// TIA Portal project "Training" (V13)

(* hardware
DEVICE "S71500/ET200MP station_1"  S7-1500 station
   slot 0: "Rail_0"  6ES7 590-1***0-0AA0
   slot 1: "PLC_1"  CPU 1516F-3 PN/DP  6ES7 516-3FN00-0AB0  V1.7
   slot 2: "DI 16x24VDC HF_1"  DI 16x24VDC HF  6ES7 521-1BH00-0AB0  V2.0
   slot 3: "AI 8xU/I/RTD/TC ST_1"  AI 8xU/I/RTD/TC ST  6ES7 531-7KF00-0AB0  V2.0
   slot 4: "CP 1543-1_1"  CP 1543-1  6GK7 543-1AX00-0XE0  V1.1
DEVICE "ET 200SP station_1"  ET 200SP-Station
   slot 0: "Rack_0"  6ES5 710-8MAx1
   slot 0: "IO device_1"  IM155-6 PN ST  6ES7 155-6AU00-0BN0  V3.1
   slot 1: "AQ 4xU/I ST_1"  AQ 4xU/I ST  6ES7 135-6HD00-0BA1  V1.0
      slot 1: "AQ 4xU/I ST_1"  AQ 4xU/I ST  6ES7 135-6HD00-0BA1
   slot 2: "DQ 16x24VDC/0.5A ST_1"  DQ 16x24VDC/0.5A ST  6ES7 132-6BH00-0BA0  V1.0
      slot 1: "DQ 16x24VDC/0.5A ST_1"  DQ 16x24VDC/0.5A ST  6ES7 132-6BH00-0BA0
   slot 3: "RQ 4x120VDC/230VAC/5A NO ST_1"  DQ 4x24VDC/2A ST  6ES7 132-6HD00-0BB0  V1.1
      slot 1: "RQ 4x120VDC/230VAC/5A NO ST_1"  RQ 4x120VDC/230VAC/5A NO ST  6ES7 132-6HD00-0BB0
   slot 4: "Server module_1"  Server module  6ES7 193-6PA00-0AA0  V1.0
      slot 1: "Server module_1"  Server module  6ES7 193-6PA00-0AA0
   slot 127: "PROFINET BusAdapter CU"  PROFINET Interface  6ES7 193-6AR00-0AA0  V0.0
      slot 1: "Port_1"  6ES7 193-6AR00-0AA0  V0.0
      slot 2: "Port_2"  6ES7 193-6AR00-0AA0  V0.0
DEVICE "KP8_1"  SIMATIC Key Panel
   slot 0: "Rack"  Rail  V1.0
   slot 0: "KP8_1"  KP8  6AV3 688-3AY36-0AX0  R01.00.00
DEVICE "S7-1200 station_1"  S7-1200 Station
   slot 0: "Rack_0"  Rack  V1.0
   slot 1: "PLC_2"  CPU 1215C AC/DC/Rly  6ES7 215-1BG40-0XB0  V4.1
*)

// ===== PLC "PLC_1"  CPU 1516F-3 PN/DP =====

VAR_GLOBAL   // PLC tag table "Default tag table"
   "System_Byte" AT %MB1 : Byte;
   "FirstScan" AT %M1.0 : Bool;
   "DiagStatusUpdate" AT %M1.1 : Bool;
   "AlwaysTRUE" AT %M1.2 : Bool;
   "AlwaysFALSE" AT %M1.3 : Bool;
   "Clock_Byte" AT %MB0 : Byte;
   "Clock_10Hz" AT %M0.0 : Bool;
   "Clock_5Hz" AT %M0.1 : Bool;
   "Clock_2.5Hz" AT %M0.2 : Bool;
   "Clock_2Hz" AT %M0.3 : Bool;
   "Clock_1.25Hz" AT %M0.4 : Bool;
   "Clock_1Hz" AT %M0.5 : Bool;
   "Clock_0.625Hz" AT %M0.6 : Bool;
   "Clock_0.5Hz" AT %M0.7 : Bool;
   "Latch Output" AT %Q50.0 : Bool;
   "Indicated Deg C_1" AT %MW2 : Int;
   "Indicated Deg c_2" AT %MW4 : Int;
   "Run Status" AT %M6.0 : Bool;
   "Counter Reset Bit" AT %M6.1 : Bool;
   "Motor 1 Running" AT %M6.2 : Bool;
   "Motor 2 Running" AT %M6.3 : Bool;
   "Outputs to Transfer Area" AT %QB100 : Byte;
   "Inputs from Transfer Area" AT %IB100 : Byte;
   "Clock Byte Data from 1200" AT %MB100 : Byte;
END_VAR

VAR_GLOBAL   // PLC tag table "Local IO Tags"
   "S71500 Green PB" AT %I0.0 : Bool;
   "S71500 Blue PB" AT %I0.1 : Bool;
   "S71500 Pot Upper" AT %IW6 : Int;
   "S71500 Pot Lower" AT %IW14 : Int;
END_VAR

VAR_GLOBAL   // PLC tag table "Remote IO Tags"
   "S7 1500 Green PB Lamp" AT %Q8.0 : Bool;
   "S7 1500 Blue PB Lamp" AT %Q8.1 : Bool;
   "1500 Demo Case Top Lights - Green" AT %Q10.0 : Bool;
   "1500 Demo Case Top Light s- Red" AT %Q10.1 : Bool;
   "1500 Demo Case Top Lights - Blue" AT %Q10.2 : Bool;
END_VAR

VAR_GLOBAL   // PLC tag table "KP8 Tags"
   "Jog_Reverse_Green_KP8" AT %Q51.5 : Bool;   // KP8
   "Enable_Disable_KP8" AT %I50.7 : Bool;   // KP8
   "Drive_Start_KP8" AT %I50.6 : Bool;   // KP8
   "Jog_Reverse_KP8" AT %I50.5 : Bool;   // KP8
   "Switch1_KP8" AT %I50.4 : Bool;   // KP8
   "Enable_Disable_Green_KP8" AT %Q51.7 : Bool;   // KP8
   "Drive_Start_Red_KP8" AT %Q50.6 : Bool;   // KP8
   "Jog_Reverse_Red_KP8" AT %Q50.5 : Bool;   // KP8
   "Switch1_Red_KP8" AT %Q50.4 : Bool;   // KP8
   "RESET_KP8" AT %I50.3 : Bool;   // KP8
   "Drive_Stop_KP8" AT %I50.2 : Bool;   // KP8
   "Jog_Forward_KP8" AT %I50.1 : Bool;   // KP8
   "RESET_Red_KP8" AT %Q50.3 : Bool;   // KP8
   "Drive_Stop_Red_KP8" AT %Q50.2 : Bool;   // KP8
   "Jog_Forward_Red_KP8" AT %Q50.1 : Bool;   // KP8
   "Switch2_KP8" AT %I50.0 : Bool;   // KP8
   "Switch2_Red_KP8" AT %Q50.0 : Bool;   // KP8
   "Enable_Disable_Red_KP8" AT %Q50.7 : Bool;   // KP8
   "Drive_Start_Green_KP8" AT %Q51.6 : Bool;   // KP8
   "Switch1_Green_KP8" AT %Q51.4 : Bool;   // KP8
   "RESET_Green_KP8" AT %Q51.3 : Bool;   // KP8
   "Drive_Stop_Green_KP8" AT %Q51.2 : Bool;   // KP8
   "Jog_Forward_Green_KP8" AT %Q51.1 : Bool;   // KP8
   "Switch2_Green_KP8" AT %Q51.0 : Bool;   // KP8
   "Switch2_Blue_KP8" AT %Q52.0 : Bool;   // KP8
   "Jog_Forward_Blue_KP8" AT %Q52.1 : Bool;   // KP8
   "Drive_Stop_Blue_KP8" AT %Q52.2 : Bool;   // KP8
   "RESET_Blue_KP8" AT %Q52.3 : Bool;   // KP8
   "Switch1_Blue_KP8" AT %Q52.4 : Bool;   // KP8
   "Jog_Reverse_Blue_KP8" AT %Q52.5 : Bool;   // KP8
   "Drive_Start_Blue_KP8" AT %Q52.6 : Bool;   // KP8
   "Enable_Disable_Blue_KP8" AT %Q52.7 : Bool;   // KP8
   "KP8_Red" AT %QB50 : Byte;   // KP8
   "KP8_Green" AT %QB51 : Byte;   // KP8
   "KP8_Blue" AT %QB52 : Byte;   // KP8
END_VAR

TYPE "Motor Control"
   STRUCT
      "Motor Start/Stop" : Bool;
      "Motor Run" : Bool;
      "Counter Reset" : Bool;
      "Count Value" : Int;
   END_STRUCT;
END_TYPE

DATA_BLOCK "My Global Data"   // DB1
{ S7_Optimized_Access := 'FALSE' }
VERSION : 0.1
   VAR
      "Celsius Temperature 1" : Int;
      "Celsius Temperature 2" : Int;
      "My INT Value" : Int;
      "My INT Setpoint Value" : Int;
   END_VAR
BEGIN
END_DATA_BLOCK

DATA_BLOCK "FB Motor Starter_DB"   // DB2
{ S7_Optimized_Access := 'FALSE' }
VERSION : 0.1
// stored: InstanceOfName FB Motor Starter
"FB Motor Starter"
BEGIN
END_DATA_BLOCK

DATA_BLOCK "FB Motor Controls_DB"   // DB3
{ S7_Optimized_Access := 'FALSE' }
VERSION : 0.1
// stored: InstanceOfName FB Motor Controls
"FB Motor Controls"
BEGIN
END_DATA_BLOCK

DATA_BLOCK "DB Motor Controls"   // DB4
{ S7_Optimized_Access := 'FALSE' }
VERSION : 0.1
   VAR
      Motor : Array[1..2] of "Motor Control";
   END_VAR
BEGIN
END_DATA_BLOCK

DATA_BLOCK "FB Motor Controls_DB_1"   // DB5
{ S7_Optimized_Access := 'FALSE' }
VERSION : 0.1
// stored: InstanceOfName FB Motor Controls
"FB Motor Controls"
BEGIN
END_DATA_BLOCK

FUNCTION_BLOCK "FB Motor Starter"   // FB1, LAD
{ S7_Optimized_Access := 'FALSE' }
VERSION : 0.1
   VAR_TEMP   // added for the SCL form of the ladder/FBD networks
      _w1 : Bool;
      _w2 : Bool;
   END_VAR
BEGIN

REGION Network 1
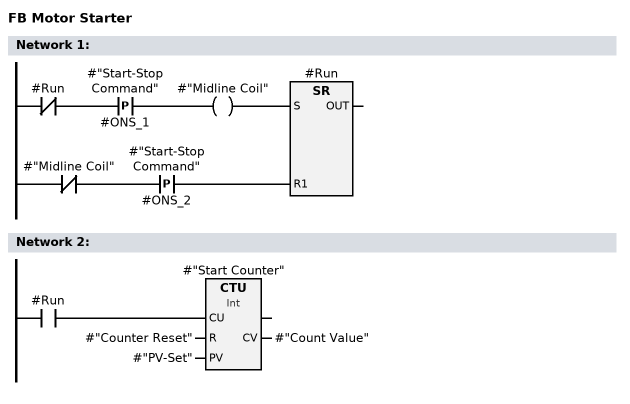
   RUNG wire#powerrail
      I_Contact( #Run )
      P_Contact(operand := #"Start-Stop Command", bit := #ONS_1)
      Coil( #"Midline Coil" )
      S_SR(operand := #Run, r1 := wire#w1)
   END_RUNG
   RUNG wire#powerrail
      I_Contact( #"Midline Coil" )
      P_Contact(operand := #"Start-Stop Command", bit := #ONS_2)
   END_RUNG wire#w1
   // the same network as SCL:
   #_w1 := NOT #Run AND #"Start-Stop Command" AND NOT #ONS_1;   // rising edge of #"Start-Stop Command"
   #ONS_1 := #"Start-Stop Command";
   #"Midline Coil" := #_w1;
   #_w2 := NOT #"Midline Coil" AND #"Start-Stop Command" AND NOT #ONS_2;   // rising edge of #"Start-Stop Command"
   #ONS_2 := #"Start-Stop Command";
   IF #_w1 THEN
       #Run := TRUE;   // SR flip-flop
   END_IF;
   IF #_w2 THEN #Run := FALSE; END_IF;
END_REGION

REGION Network 2
   #"Start Counter".CTU(CU := #Run, R := #"Counter Reset", PV := #"PV-Set", CV => #"Count Value");
END_REGION
END_FUNCTION_BLOCK

FUNCTION_BLOCK "FB Motor Controls"   // FB2, LAD
{ S7_Optimized_Access := 'FALSE' }
VERSION : 0.1
BEGIN

REGION Network 1
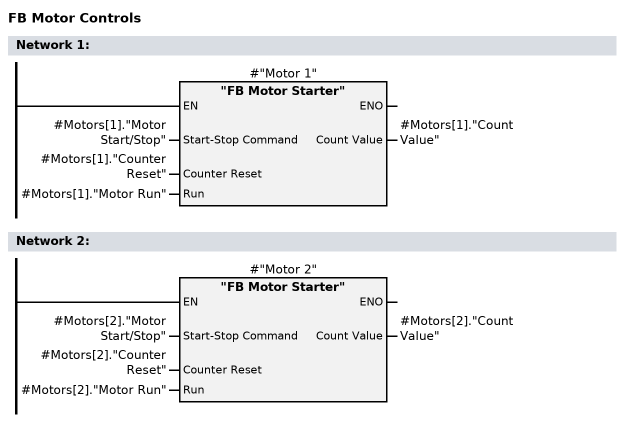
   RUNG wire#powerrail
      #"Motor 1"("Start-Stop Command" := #Motors[1]."Motor Start/Stop", "Counter Reset" := #Motors[1]."Counter Reset", Run := #Motors[1]."Motor Run", "Count Value" => #Motors[1]."Count Value")
   END_RUNG
   // the same network as SCL:
   #"Motor 1"("Start-Stop Command" := #Motors[1]."Motor Start/Stop",   // "FB Motor Starter"
              "Counter Reset" := #Motors[1]."Counter Reset",
              Run := #Motors[1]."Motor Run",
              "Count Value" => #Motors[1]."Count Value");
END_REGION

REGION Network 2
   RUNG wire#powerrail
      #"Motor 2"("Start-Stop Command" := #Motors[2]."Motor Start/Stop", "Counter Reset" := #Motors[2]."Counter Reset", Run := #Motors[2]."Motor Run", "Count Value" => #Motors[2]."Count Value")
   END_RUNG
   // the same network as SCL:
   #"Motor 2"("Start-Stop Command" := #Motors[2]."Motor Start/Stop",   // "FB Motor Starter"
              "Counter Reset" := #Motors[2]."Counter Reset",
              Run := #Motors[2]."Motor Run",
              "Count Value" => #Motors[2]."Count Value");
END_REGION
END_FUNCTION_BLOCK

FUNCTION "F to C Conversion" : Void   // FC1, LAD
{ S7_Optimized_Access := 'FALSE' }
VERSION : 0.1
BEGIN

REGION Network 1
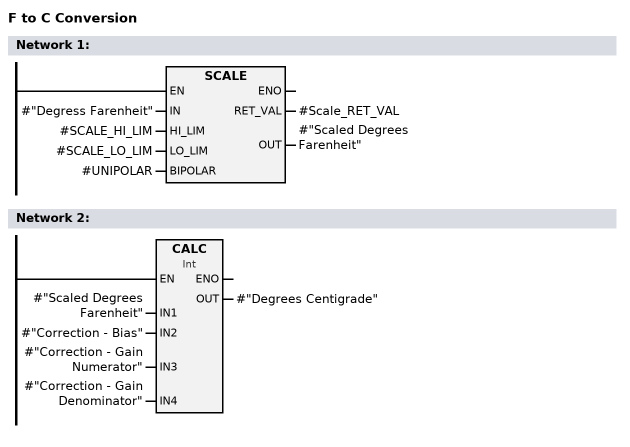
   #Scale_RET_VAL := SCALE(IN := #"Degress Farenheit",
                           HI_LIM := #SCALE_HI_LIM,
                           LO_LIM := #SCALE_LO_LIM,
                           BIPOLAR := #UNIPOLAR,
                           OUT => #"Scaled Degrees Farenheit");
END_REGION

REGION Network 2
   CALC(in1 := #"Scaled Degrees Farenheit",
        in2 := #"Correction - Bias",
        in3 := #"Correction - Gain Numerator",
        in4 := #"Correction - Gain Denominator",
        out => #"Degrees Centigrade");
END_REGION
END_FUNCTION

ORGANIZATION_BLOCK "Main"   // OB1, LAD, ProgramCycle
TITLE = "Main Program Sweep (Cycle)"
{ S7_Optimized_Access := 'FALSE' }
VERSION : 0.1
BEGIN

REGION Network 1
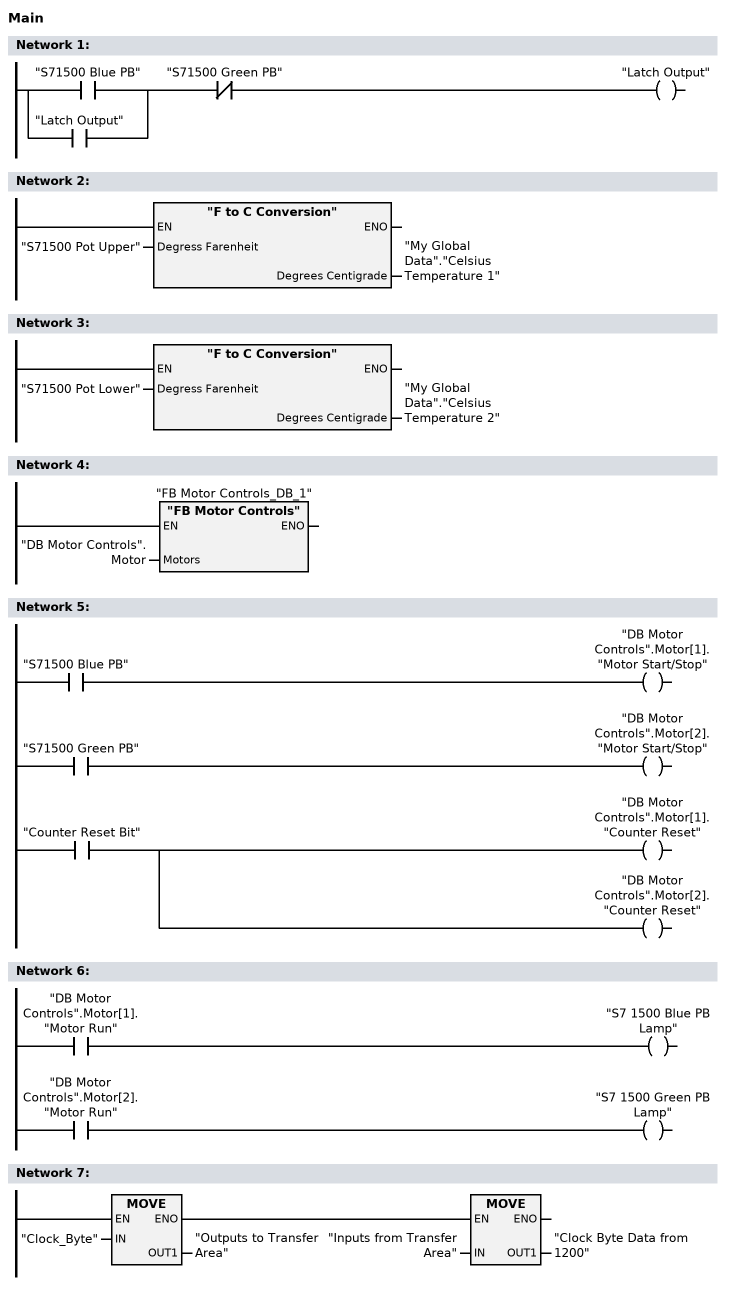
   RUNG wire#powerrail
      Contact( "S71500 Blue PB" )
      wire#w1
      I_Contact( "S71500 Green PB" )
      Coil( "Latch Output" )
   END_RUNG
   RUNG wire#powerrail
      Contact( "Latch Output" )
   END_RUNG wire#w1
   // the same network as SCL:
   "Latch Output" := ("S71500 Blue PB" OR "Latch Output") AND NOT "S71500 Green PB";
END_REGION

REGION Network 2
   RUNG wire#powerrail
      "F to C Conversion"("Degress Farenheit" := "S71500 Pot Upper", "Degrees Centigrade" => "My Global Data"."Celsius Temperature 1")
   END_RUNG
   // the same network as SCL:
   "F to C Conversion"("Degress Farenheit" := "S71500 Pot Upper",
                       "Degrees Centigrade" => "My Global Data"."Celsius Temperature 1");
END_REGION

REGION Network 3
   RUNG wire#powerrail
      "F to C Conversion"("Degress Farenheit" := "S71500 Pot Lower", "Degrees Centigrade" => "My Global Data"."Celsius Temperature 2")
   END_RUNG
   // the same network as SCL:
   "F to C Conversion"("Degress Farenheit" := "S71500 Pot Lower",
                       "Degrees Centigrade" => "My Global Data"."Celsius Temperature 2");
END_REGION

REGION Network 4
   RUNG wire#powerrail
      "FB Motor Controls_DB_1"(Motors := "DB Motor Controls".Motor)
   END_RUNG
   // the same network as SCL:
   "FB Motor Controls_DB_1"(Motors := "DB Motor Controls".Motor);   // "FB Motor Controls"
END_REGION

REGION Network 5
   RUNG wire#powerrail
      Contact( "S71500 Blue PB" )
      Coil( "DB Motor Controls".Motor[1]."Motor Start/Stop" )
   END_RUNG
   RUNG wire#powerrail
      Contact( "S71500 Green PB" )
      Coil( "DB Motor Controls".Motor[2]."Motor Start/Stop" )
   END_RUNG
   RUNG wire#powerrail
      Contact( "Counter Reset Bit" )
      wire#w1
      Coil( "DB Motor Controls".Motor[1]."Counter Reset" )
   END_RUNG
   RUNG wire#w1
      Coil( "DB Motor Controls".Motor[2]."Counter Reset" )
   END_RUNG
   // the same network as SCL:
   "DB Motor Controls".Motor[1]."Motor Start/Stop" := "S71500 Blue PB";
   "DB Motor Controls".Motor[2]."Motor Start/Stop" := "S71500 Green PB";
   "DB Motor Controls".Motor[1]."Counter Reset" := "Counter Reset Bit";
   "DB Motor Controls".Motor[2]."Counter Reset" := "Counter Reset Bit";
END_REGION

REGION Network 6
   RUNG wire#powerrail
      Contact( "DB Motor Controls".Motor[1]."Motor Run" )
      Coil( "S7 1500 Blue PB Lamp" )
   END_RUNG
   RUNG wire#powerrail
      Contact( "DB Motor Controls".Motor[2]."Motor Run" )
      Coil( "S7 1500 Green PB Lamp" )
   END_RUNG
   // the same network as SCL:
   "S7 1500 Blue PB Lamp" := "DB Motor Controls".Motor[1]."Motor Run";
   "S7 1500 Green PB Lamp" := "DB Motor Controls".Motor[2]."Motor Run";
END_REGION

REGION Network 7
   RUNG wire#powerrail
      Move(in := "Clock_Byte", out1 => "Outputs to Transfer Area")
      Move(in := "Inputs from Transfer Area", out1 => "Clock Byte Data from 1200")
   END_RUNG
   // the same network as SCL:
   "Outputs to Transfer Area" := "Clock_Byte";
   "Clock Byte Data from 1200" := "Inputs from Transfer Area";
END_REGION
END_ORGANIZATION_BLOCK

// ===== PLC "PLC_2"  CPU 1215C AC/DC/Rly =====

VAR_GLOBAL   // PLC tag table "Default tag table"
   "System_Byte" AT %MB1 : Byte;
   "FirstScan" AT %M1.0 : Bool;
   "DiagStatusUpdate" AT %M1.1 : Bool;
   "AlwaysTRUE" AT %M1.2 : Bool;
   "AlwaysFALSE" AT %M1.3 : Bool;
   "Clock_Byte" AT %MB0 : Byte;
   "Clock_10Hz" AT %M0.0 : Bool;
   "Clock_5Hz" AT %M0.1 : Bool;
   "Clock_2.5Hz" AT %M0.2 : Bool;
   "Clock_2Hz" AT %M0.3 : Bool;
   "Clock_1.25Hz" AT %M0.4 : Bool;
   "Clock_1Hz" AT %M0.5 : Bool;
   "Clock_0.625Hz" AT %M0.6 : Bool;
   "Clock_0.5Hz" AT %M0.7 : Bool;
   "Inputs from Transfer Area" AT %IB100 : Byte;
   "Outputs to Transfer Area" AT %QB100 : Byte;
   "Clock Byte Data from S7 1500" AT %MB100 : Byte;
END_VAR

ORGANIZATION_BLOCK "Main"   // OB1, LAD, ProgramCycle
TITLE = "Main Program Sweep (Cycle)"
{ S7_Optimized_Access := 'FALSE' }
VERSION : 0.1
BEGIN

REGION Network 1
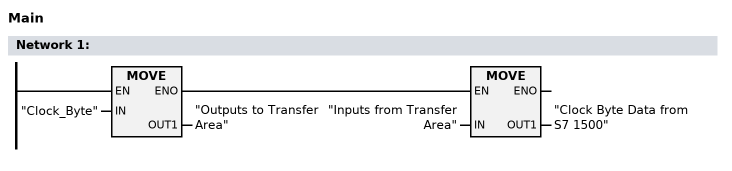
   RUNG wire#powerrail
      Move(in := "Clock_Byte", out1 => "Outputs to Transfer Area")
      Move(in := "Inputs from Transfer Area", out1 => "Clock Byte Data from S7 1500")
   END_RUNG
   // the same network as SCL:
   "Outputs to Transfer Area" := "Clock_Byte";
   "Clock Byte Data from S7 1500" := "Inputs from Transfer Area";
END_REGION
END_ORGANIZATION_BLOCK